TYPE DUT_Motor_Freq :
STRUCT
	Cs: DUT_CS_Valve;
	Hmi: DUT_HMI_Valve;
	Sts: DUT_STS_Valve;
	Alm: DUT_ALM_Valve;
END_STRUCT
END_TYPE

(* stored: Version 1.1.0.1, ProductVersion 3.1.4024.12
   DUT DUT_Motor_Freq: Id {9d20675a-7e91-401d-a1df-5325fb26f757} *)
